Staubli VAL3: actGesture.pgx

program actGesture()
begin
  //putln("GestureCalled")
  //putln(sInput)
  if (sInput=="fist")
    call gestureFist()
  elseIf (sInput=="waveIn")
    call gestureWaveIn()
  elseIf (sInput=="waveOut")
    call gestureWaveout()
  elseIf (sInput=="fingersSpread")
    call gestureSpread()
  endIf

end
